# EPICS autosave request: apps/iocBoot/iocclassc1test/joerger_classc1_settings.req
#
# Call once per scaler.  Should match associated substitutions file.
#
# Requires: set_requestfile_path for std and calc
#   set_requestfile_path(calc,     "calcApp/Db")
#   set_requestfile_path(std,      "stdApp/Db")
#
file "joerger_settings.req", P=scaler,  S=_c
file "joerger_settings.req", P=scaler,  S=_d
file "joerger_settings.req", P=scaler,  S=_e
